// TIA Portal V19 export
TYPE "typeAxisControlMaintenance"
// stored: Access Published
   STRUCT
      upperVel : LReal := 100.0;   // 维护速度上限
      vel : LReal := 20.0;   // 维护速度设定值，画面做限制根据上限值如果超了不允许输入
      acc : LReal := 2.0;
      dec : LReal := 2.0;
   END_STRUCT;
END_TYPE
